FUNCTION_BLOCK FB_Door_Closed
VAR_INPUT
	valve																: BOOL;
	limit_switch														: BOOL;
END_VAR
VAR_OUTPUT
	door_closed															: BOOL;
END_VAR
VAR
	ton1																: TON;
	rtrig1																: R_TRIG;
END_VAR

// FB_Door_Closed
// Rev 1.0 - November 2, 2024

ton1(IN:= valve AND limit_switch, PT:= _DOOR_LATCH_CLOSE_TIME);
rtrig1(CLK:= ton1.Q);
IF rtrig1.Q THEN
	door_closed															:= TRUE;
ELSIF NOT valve THEN
	door_closed															:= FALSE;
END_IF

END_FUNCTION_BLOCK

(* stored: Version 1.1.0.1, ProductVersion 3.1.4024.13
   POU FB_Door_Closed: Id {30508aa0-fc69-4a73-937d-a80ff2cb8d53}, SpecialFunc None *)
